// TIA Portal project "s71200_modbus_config" (V16)
// Modbus main program for S7-1200. Use with scada_app.py and plant_app.py.

(* hardware
DEVICE "S7-1200 station_1"  S7-1200 Station
   slot 0: "Rack_0"  S7-1200 Rack  Rack  V1.0
   slot 1: "quicksilver"  CPU 1211C DC/DC/DC  6ES7 211-1AE40-0XB0  V4.4
*)

// ===== PLC "quicksilver"  CPU 1211C DC/DC/DC =====

VAR_GLOBAL   // PLC tag table "Default tag table"
   "System_Byte" AT %MB1 : Byte;
   "FirstScan" AT %M1.0 : Bool;
   "DiagStatusUpdate" AT %M1.1 : Bool;
   "AlwaysTRUE" AT %M1.2 : Bool;
   "AlwaysFALSE" AT %M1.3 : Bool;
   "Clock_Byte" AT %MB0 : Byte;
   "Clock_10Hz" AT %M0.0 : Bool;
   "Clock_5Hz" AT %M0.1 : Bool;
   "Clock_2.5Hz" AT %M0.2 : Bool;
   "Clock_2Hz" AT %M0.3 : Bool;
   "Clock_1.25Hz" AT %M0.4 : Bool;
   "Clock_1Hz" AT %M0.5 : Bool;
   "Clock_0.625Hz" AT %M0.6 : Bool;
   "Clock_0.5Hz" AT %M0.7 : Bool;
   "dc_input_I0" AT %IW0 : Int;
   "ain_0" AT %IW64 : Int;   // Analog input 1 - red from LJ
   "ain_1" AT %IW66 : Int;   // Analog input 2 - orange form LJ
   "aout_1" AT %QW1 : Int;
   "error_ainput" AT %Q0.3 : Bool;
   "temp_signal1" AT %MW70 : Int;
   "temp_out" AT %MW72 : Int;
   "led_q0" AT %Q0.0 : Bool;
   "led_q1" AT %Q0.1 : Bool;
   "temp_base" AT %MW74 : Int;   // Temp copy
   "signal1" AT %MW76 : Int;
   "signal2" AT %MW78 : Int;
   "offset" AT %MW80 : Int;
   "temp_signal2" AT %MW82 : Int;
   "aout_0" AT %QW0 : Int;
END_VAR

DATA_BLOCK "modbus_config_server"   // DB2
{ S7_Optimized_Access := 'TRUE' }
VERSION : 0.1
   VAR
      DISCONNECT : Bool;
      CONNECT : TCON_IP_v4;
      DR : Bool;
      NDR : Bool;
      ERROR : Bool;
      STATUS : Word;
   END_VAR
BEGIN
   CONNECT.ConnectionType := 11;
   CONNECT.ID := 1;
   CONNECT.InterfaceId := 64;
   CONNECT.LocalPort := 502;
END_DATA_BLOCK

DATA_BLOCK "modbus_buffer_server"   // DB3
{ S7_Optimized_Access := 'TRUE' }
VERSION : 0.1
   VAR
      BUFFER : Array[0..63] of Int;
   END_VAR
BEGIN
END_DATA_BLOCK

FUNCTION "analog_input_0-10v" : Void   // FC1, LAD
{ S7_Optimized_Access := 'TRUE' }
VERSION : 0.1
   VAR_INPUT
      "Input_Channel_0-10v" : Int;
      Lower_Value : Int;
      Upper_Value : Int;
   END_VAR
   VAR_OUTPUT
      Output_Value : Real;
      Error : Bool;
   END_VAR
   VAR_TEMP
      Temp1 : Real;
   END_VAR
BEGIN

REGION Network 1
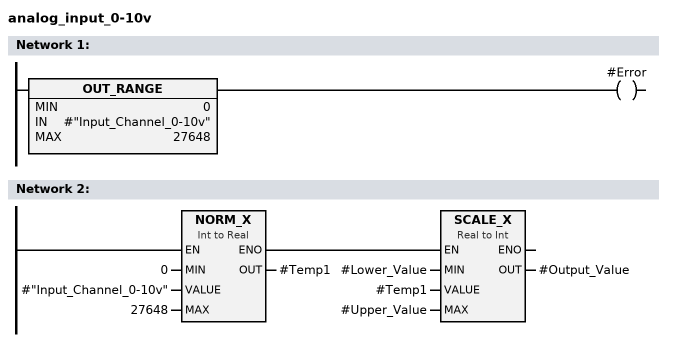
   #Error := (#"Input_Channel_0-10v" < 0) OR (#"Input_Channel_0-10v" > 27648);
END_REGION

REGION Network 2
   RUNG wire#powerrail
      { S7_Templates := "[SrcType := Int, DestType := Real]" } Normalize(min := 0, value := #"Input_Channel_0-10v", max := 27648, out => #Temp1)
      { S7_Templates := "[SrcType := Real, DestType := Int]" } Scale(min := #Lower_Value, value := #Temp1, max := #Upper_Value, out => #Output_Value)
   END_RUNG
   // the same network as SCL:
   #Temp1 := NORM_X(MIN := 0, VALUE := #"Input_Channel_0-10v", MAX := 27648);
   #Output_Value := SCALE_X(MIN := #Lower_Value, VALUE := #Temp1, MAX := #Upper_Value);
END_REGION
END_FUNCTION

ORGANIZATION_BLOCK "main_modbus"   // OB1, LAD, ProgramCycle
TITLE = "Main Program Sweep (Cycle)"
{ S7_Optimized_Access := 'TRUE' }
VERSION : 0.1
   VAR_INPUT
      Initial_Call : Bool;   // Initial call of this OB
      Remanence : Bool;   // =True, if remanent data are available
   END_VAR
   VAR_TEMP   // added for the SCL form of the ladder/FBD networks
      _w1 : Bool;
      _w2 : Bool;
   END_VAR
BEGIN

REGION Network 1: Modbus Communication
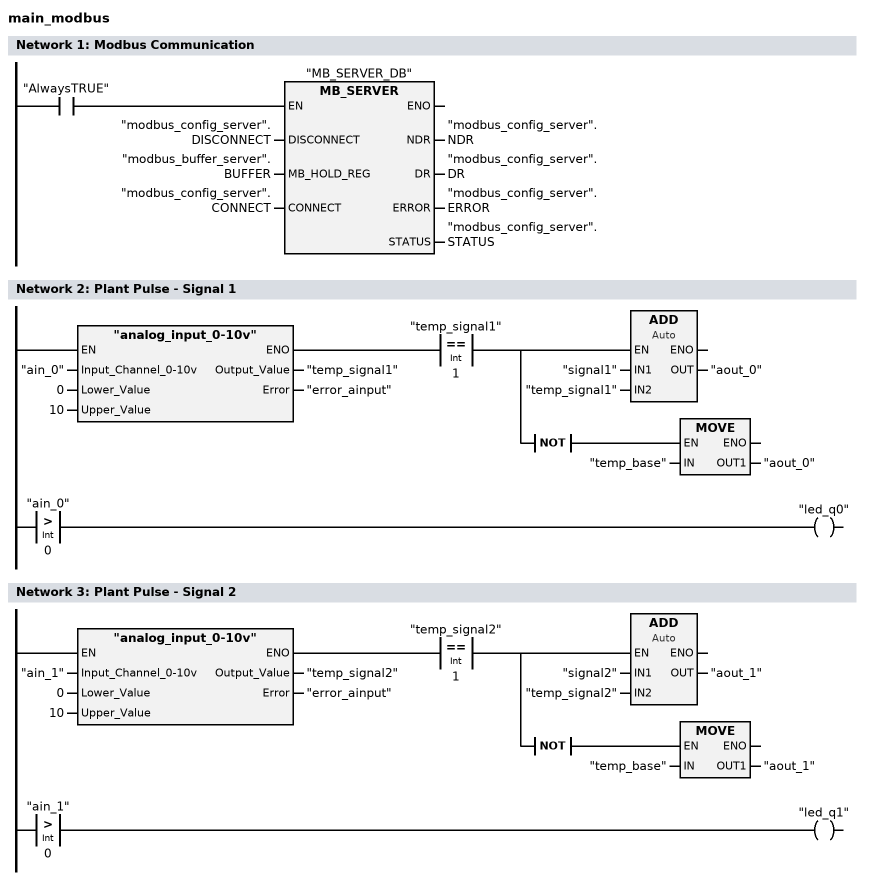
   IF "AlwaysTRUE" THEN
       "MB_SERVER_DB"(DISCONNECT := "modbus_config_server".DISCONNECT,   // MB_SERVER
                      MB_HOLD_REG := "modbus_buffer_server".BUFFER,
                      CONNECT := "modbus_config_server".CONNECT,
                      NDR => "modbus_config_server".NDR,
                      DR => "modbus_config_server".DR,
                      ERROR => "modbus_config_server".ERROR,
                      STATUS => "modbus_config_server".STATUS);
   END_IF;
END_REGION

REGION Network 2: Plant Pulse - Signal 1
   RUNG wire#powerrail
      "analog_input_0-10v"("Input_Channel_0-10v" := "ain_0", Lower_Value := 0, Upper_Value := 10, Output_Value => "temp_signal1", Error => "error_ainput")
      { S7_Templates := "SrcType := Int" } EQ_Contact(in1 := "temp_signal1", in2 := 1)
      wire#w1
      Add(in1 := "signal1", in2 := "temp_signal1", out => "aout_0")
   END_RUNG
   RUNG wire#w1
      Not()
      Move(in := "temp_base", out1 => "aout_0")
   END_RUNG
   RUNG wire#powerrail
      { S7_Templates := "SrcType := Int" } GT_Contact(in1 := "ain_0", in2 := 0)
      Coil( "led_q0" )
   END_RUNG
   // the same network as SCL:
   "analog_input_0-10v"("Input_Channel_0-10v" := "ain_0",
                        Lower_Value := 0,
                        Upper_Value := 10,
                        Output_Value => "temp_signal1",
                        Error => "error_ainput",
                        ENO => #_w1);
   #_w2 := #_w1 AND ("temp_signal1" = 1);
   IF #_w2 THEN "aout_0" := "signal1" + "temp_signal1"; END_IF;
   IF NOT #_w2 THEN "aout_0" := "temp_base"; END_IF;
   "led_q0" := "ain_0" > 0;
END_REGION

REGION Network 3: Plant Pulse - Signal 2
   RUNG wire#powerrail
      "analog_input_0-10v"("Input_Channel_0-10v" := "ain_1", Lower_Value := 0, Upper_Value := 10, Output_Value => "temp_signal2", Error => "error_ainput")
      { S7_Templates := "SrcType := Int" } EQ_Contact(in1 := "temp_signal2", in2 := 1)
      wire#w1
      Add(in1 := "signal2", in2 := "temp_signal2", out => "aout_1")
   END_RUNG
   RUNG wire#w1
      Not()
      Move(in := "temp_base", out1 => "aout_1")
   END_RUNG
   RUNG wire#powerrail
      { S7_Templates := "SrcType := Int" } GT_Contact(in1 := "ain_1", in2 := 0)
      Coil( "led_q1" )
   END_RUNG
   // the same network as SCL:
   "analog_input_0-10v"("Input_Channel_0-10v" := "ain_1",
                        Lower_Value := 0,
                        Upper_Value := 10,
                        Output_Value => "temp_signal2",
                        Error => "error_ainput",
                        ENO => #_w1);
   #_w2 := #_w1 AND ("temp_signal2" = 1);
   IF #_w2 THEN "aout_1" := "signal2" + "temp_signal2"; END_IF;
   IF NOT #_w2 THEN "aout_1" := "temp_base"; END_IF;
   "led_q1" := "ain_1" > 0;
END_REGION
END_ORGANIZATION_BLOCK

ORGANIZATION_BLOCK "temp_holder"   // OB123, LAD, ProgramCycle
TITLE = "Main Program Sweep (Cycle)"
{ S7_Optimized_Access := 'TRUE' }
VERSION : 0.1
   VAR_INPUT
      Initial_Call : Bool;   // Initial call of this OB
      Remanence : Bool;   // =True, if remanent data are available
   END_VAR
   VAR_TEMP   // added for the SCL form of the ladder/FBD networks
      _w1 : Bool;
      _w2 : Bool;
   END_VAR
BEGIN

REGION Network 1: Plant Pulse - offset setter
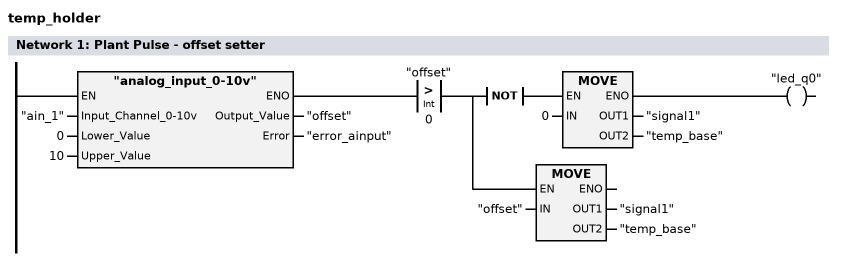
   RUNG wire#powerrail
      "analog_input_0-10v"("Input_Channel_0-10v" := "ain_1", Lower_Value := 0, Upper_Value := 10, Output_Value => "offset", Error => "error_ainput")
      { S7_Templates := "SrcType := Int" } GT_Contact(in1 := "offset", in2 := 0)
      wire#w1
      Not()
      Move(in := 0, out1 => "signal1", out2 => "temp_base")
      Coil( "led_q0" )
   END_RUNG
   RUNG wire#w1
      Move(in := "offset", out1 => "signal1", out2 => "temp_base")
   END_RUNG
   // the same network as SCL:
   "analog_input_0-10v"("Input_Channel_0-10v" := "ain_1",
                        Lower_Value := 0,
                        Upper_Value := 10,
                        Output_Value => "offset",
                        Error => "error_ainput",
                        ENO => #_w1);
   #_w2 := #_w1 AND ("offset" > 0);
   IF NOT #_w2 THEN
       "signal1" := 0;
       "temp_base" := 0;
   END_IF;
   "led_q0" := NOT #_w2;
   IF #_w2 THEN
       "signal1" := "offset";
       "temp_base" := "offset";
   END_IF;
END_REGION
END_ORGANIZATION_BLOCK